// TIA Portal V17 export
// export: Created 2022-10-14T12:26:29.2830673Z, ExportSetting WithDefaults, DisplayName Totally Integrated Automation Portal, DisplayVersion V17 Update 4, DisplayName TIA Portal Openness, DisplayVersion V17 Update 4, DisplayName TIA Portal Version Control Interface, DisplayVersion V17, DisplayName SINAMICS Startdrive Advanced, DisplayVersion V17 Update2, DisplayName SINAMICS Startdrive G130, G150, S120, S150, SINAMICS MV, S210, DisplayVersion V17 Update2, DisplayName SINAMICS Startdrive G110M, G120, G120C, G120D, G120P, G115D, DisplayVersion V17 Update2, DisplayName STEP 7 Professional, DisplayVersion V17 Update 4, DisplayName STEP 7 Safety, DisplayVersion V17, DisplayName WinCC Advanced / Unified PC, DisplayVersion V17 Update 4
FUNCTION_BLOCK "SITOP_PSE200U"   // FB8700, FBD
{ S7_Optimized_Access := 'TRUE' }
VERSION : 0.1
// stored: AutoNumber false, IsIECCheckEnabled false, IsRetainMemResEnabled false, MemoryReserve 100, SetENOAutomatically false, UDAEnableTagReadback false
   VAR_INPUT
      Status_Signal : Bool;
   END_VAR
   VAR_OUTPUT
      Out_1 : Bool;
      Out_2 : Bool;
      Out_3 : Bool;
      Out_4 : Bool;
   END_VAR
   VAR
      IEC_Timer_1 { S7_SetPoint := 'True'} : TON_TIME;
      zyklus : Time;
      SR2 : Bool;
      SR3 : Bool;
      SR4 : Bool;
      SR5 : Bool;
      HM1 : Bool;
   END_VAR
BEGIN

REGION Network 1: Ermitteln START Flanke
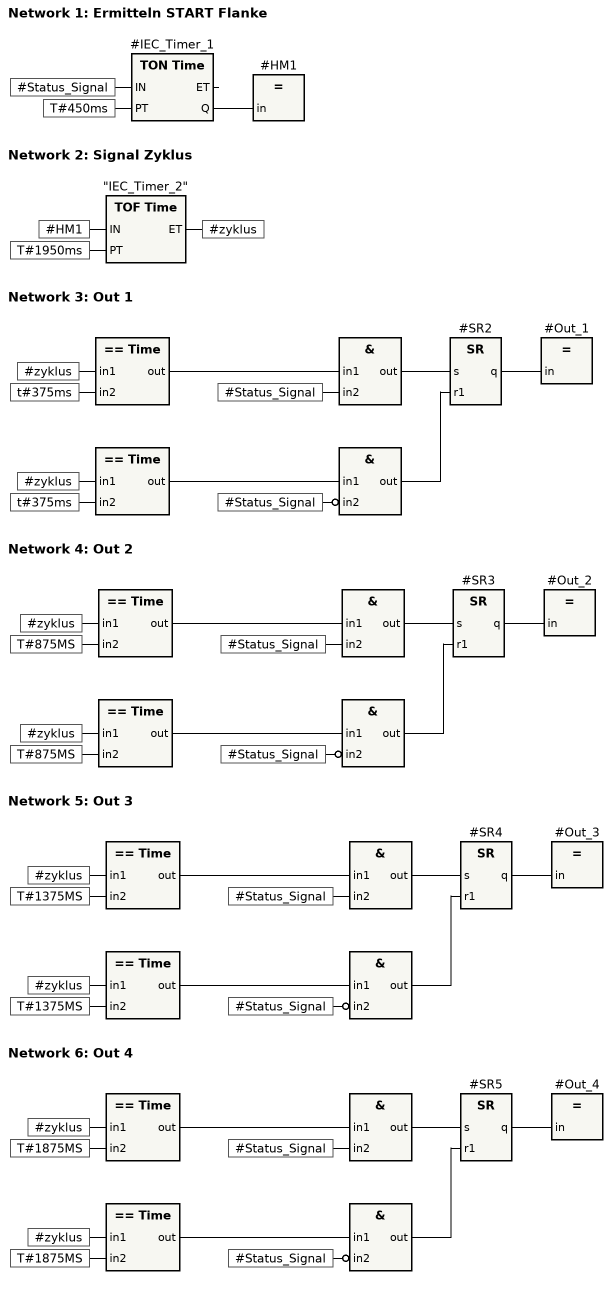
   #IEC_Timer_1(IN := #Status_Signal, PT := T#450ms);   // TON
   #HM1 := #IEC_Timer_1.Q;
END_REGION

REGION Network 2: Signal Zyklus
   "IEC_Timer_2".TOF(IN := #HM1, PT := T#1950ms, ET => #zyklus);
END_REGION

REGION Network 3: Out 1
   IF (#zyklus = t#375ms) AND #Status_Signal THEN
       #SR2 := TRUE;   // SR flip-flop
   END_IF;
   IF (#zyklus = t#375ms) AND NOT #Status_Signal THEN #SR2 := FALSE; END_IF;
   #Out_1 := #SR2;
END_REGION

REGION Network 4: Out 2
   IF (#zyklus = T#875MS) AND #Status_Signal THEN
       #SR3 := TRUE;   // SR flip-flop
   END_IF;
   IF (#zyklus = T#875MS) AND NOT #Status_Signal THEN #SR3 := FALSE; END_IF;
   #Out_2 := #SR3;
END_REGION

REGION Network 5: Out 3
   IF (#zyklus = T#1375MS) AND #Status_Signal THEN
       #SR4 := TRUE;   // SR flip-flop
   END_IF;
   IF (#zyklus = T#1375MS) AND NOT #Status_Signal THEN #SR4 := FALSE; END_IF;
   #Out_3 := #SR4;
END_REGION

REGION Network 6: Out 4
   IF (#zyklus = T#1875MS) AND #Status_Signal THEN
       #SR5 := TRUE;   // SR flip-flop
   END_IF;
   IF (#zyklus = T#1875MS) AND NOT #Status_Signal THEN #SR5 := FALSE; END_IF;
   #Out_4 := #SR5;
END_REGION
END_FUNCTION_BLOCK
